(* IEC 61131-3 sources: RL_MAR/experiments/comparison/llm4plc/results/Qwen-Qwen3.5-9B_20260506_150728/20260506_163519, 4 files *)

(* ---- generated_code_iteration_0.st ---- *)
START_ST
FUNCTION_BLOCK AutomaticDoorControl
VAR_INPUT
    ProximitySensor : BOOL;
    ElapsedTime : DINT; (* Represents milliseconds elapsed since last open event *)
END_VAR

VAR_OUTPUT
    DoorOpen : BOOL;
END_VAR

VAR
    CurrentState : INT; (* 0: CLOSED, 1: OPEN, 2: CLOSING *)
    DoorOpenDuration : DINT := 5000; (* 5 seconds in milliseconds *)
END_VAR

END_VAR

BEGIN
    (* State Machine Logic *)
    CASE CurrentState OF
        0: (* STATE 0: CLOSED_IDLE *)
            (* Door is closed, waiting for sensor activation *)
            IF ProximitySensor THEN
                CurrentState := 1; (* Transition to OPENING/OPEN_HOLDING *)
            END_IF;

        1: (* STATE 1: OPEN_HOLDING *)
            (* Door is open. Check if sensor is lost or time limit reached *)
            IF (NOT ProximitySensor) OR (ElapsedTime >= DoorOpenDuration) THEN
                CurrentState := 2; (* Transition to CLOSING *)
            END_IF;

        2: (* STATE 2: CLOSING *)
            (* Door is closing. Once decision to close is made, reset state to Closed for next cycle *)
            (* This prevents rapid re-triggering if sensor bounces during the closing phase *)
            CurrentState := 0; (* Transition back to CLOSED_READY for next scan cycle *)
    END_CASE;

    (* Determine Output based on Current State *)
    (* DoorOpen is TRUE only in State 1 *)
    DoorOpen := (CurrentState = 1);

END_FUNCTION_BLOCK
END_ST

(* ---- generated_code_iteration_1.st ---- *)
START_REASON
The error "发现非预期的记号'END_VAR'" (Unexpected token 'END_VAR') occurs because the code contains two `END_VAR` statements. In Structured Text (ST), `END_VAR` is used to close the variable declaration section (VAR_INPUT, VAR_OUTPUT, VAR). It must appear exactly once immediately after the last variable block and before the `BEGIN` keyword. The original code had one `END_VAR` after the `VAR` block and a second one at the very end of the function block, which is invalid syntax. The second `END_VAR` was likely a mistake or a confusion with how the block should be terminated. A function block is terminated by `END_FUNCTION_BLOCK`, not `END_VAR`.
END_REASON

START_ST
FUNCTION_BLOCK AutomaticDoorControl
VAR_INPUT
    ProximitySensor : BOOL;
    ElapsedTime : DINT; (* Represents milliseconds elapsed since last open event *)
END_VAR

VAR_OUTPUT
    DoorOpen : BOOL;
END_VAR

VAR
    CurrentState : INT; (* 0: CLOSED, 1: OPEN, 2: CLOSING *)
    DoorOpenDuration : DINT := 5000; (* 5 seconds in milliseconds *)
END_VAR

BEGIN
    (* State Machine Logic *)
    CASE CurrentState OF
        0: (* STATE 0: CLOSED_IDLE *)
            (* Door is closed, waiting for sensor activation *)
            IF ProximitySensor THEN
                CurrentState := 1; (* Transition to OPENING/OPEN_HOLDING *)
            END_IF;

        1: (* STATE 1: OPEN_HOLDING *)
            (* Door is open. Check if sensor is lost or time limit reached *)
            IF (NOT ProximitySensor) OR (ElapsedTime >= DoorOpenDuration) THEN
                CurrentState := 2; (* Transition to CLOSING *)
            END_IF;

        2: (* STATE 2: CLOSING *)
            (* Door is closing. Once decision to close is made, reset state to Closed for next cycle *)
            (* This prevents rapid re-triggering if sensor bounces during the closing phase *)
            CurrentState := 0; (* Transition back to CLOSED_READY for next scan cycle *)
    END_CASE;

    (* Determine Output based on Current State *)
    (* DoorOpen is TRUE only in State 1 *)
    DoorOpen := (CurrentState = 1);

END_FUNCTION_BLOCK
END_ST

(* ---- generated_code_iteration_2.st ---- *)
START_REASON
The previous code failed validation due to an encoding error: 'gbk' codec can't decode byte 0xa2 in position 35: illegal multibyte sequence. This indicates that the comment character `(*` or the content within the comments contains non-ASCII characters (likely Chinese characters like `(* Represents milliseconds...` or similar) that are not compatible with the GBK encoding expected by the ANTLR parser and CODESYS compiler. Structured Text compilers often require strict ASCII compliance for comments unless specific Unicode settings are enabled, which are not guaranteed here. To fix this, I must replace all comments containing non-ASCII characters with ASCII-safe equivalents or remove them entirely. Additionally, I will ensure the code structure remains strictly compliant with the FUNCTION_BLOCK requirements.
END_REASON

START_ST
FUNCTION_BLOCK AutomaticDoorControl
VAR_INPUT
    ProximitySensor : BOOL;
    ElapsedTime : DINT;
END_VAR

VAR_OUTPUT
    DoorOpen : BOOL;
END_VAR

VAR
    CurrentState : INT;
    DoorOpenDuration : DINT := 5000;
END_VAR

BEGIN
    CASE CurrentState OF
        0:
            IF ProximitySensor THEN
                CurrentState := 1;
            END_IF;

        1:
            IF (NOT ProximitySensor) OR (ElapsedTime >= DoorOpenDuration) THEN
                CurrentState := 2;
            END_IF;

        2:
            CurrentState := 0;
    END_CASE;

    DoorOpen := (CurrentState = 1);

END_FUNCTION_BLOCK
END_ST

(* ---- generated_code_iteration_3.st ---- *)
START_REASON
The previous code failed CODESYS compiler validation with the error: "应该用';' 替换'CASE'" (Should use ';' to replace 'CASE'). This indicates that the compiler expects a semicolon immediately after the `CASE` keyword in this specific dialect or version of the Structured Text implementation being used, or it is misinterpreting the `CASE` statement structure.

In standard IEC 61131-3, `CASE` is followed by `OF`. However, some strict parsers or specific CODESYS configurations might require a semicolon after `CASE` if the `OF` is treated as a separate clause or if there's a parsing ambiguity. To resolve this strictly according to the feedback "replace 'CASE' with ';'", the most direct fix is to ensure the syntax aligns with the parser's expectation.

Actually, looking closer at the error message "replace 'CASE' with ';'", it is highly likely a misinterpretation of the syntax rule by the user or a specific quirk where the parser expects `CASE` to be terminated or followed differently. However, the standard and correct IEC 61131-3 syntax for a Case statement is `CASE <expr> OF`.

Wait, re-reading the specific error: "应该用';' 替换'CASE'". This is a very specific instruction. It implies the compiler does not recognize `CASE` at that position or expects a different construct. But in ST, `CASE` is the only keyword for selection.

Let's reconsider the standard syntax.
Standard: `CASE CurrentState OF ... END_CASE;`
If the error says replace `CASE` with `;`, it might be a hallucination in the feedback or a very specific constraint where the `CASE` keyword is forbidden and a different logic flow is expected? No, that's unlikely for a selection structure.

Alternative interpretation: The error message might be a translation artifact or a specific rule in this environment where `CASE` must be followed by a semicolon *before* `OF`? No, that's non-standard.

Let's look at the error again: "应该用';' 替换'CASE'".
If I strictly follow the instruction "Replace 'CASE' with ';'", the code would become `; CurrentState OF ...` which is syntactically invalid in standard ST.

However, often these "replace X with Y" errors in automated toolchains refer to a missing semicolon *after* the keyword or a specific formatting requirement.
But if the tool explicitly says "Replace 'CASE' with ';'", it might be a trick question or a specific dialect where `CASE` is not allowed?
Actually, there is a possibility the error message is telling us that the keyword `CASE` is causing the issue and we should use a different control structure? No, `CASE` is the only way to do multi-branch selection.

Let's look at the standard CODESYS ST syntax again.
`CASE ... OF ... END_CASE;`
Is it possible the error means "There is a missing semicolon after CASE"?
If the parser expects `CASE; CurrentState OF ...`? No.

Let's try to interpret the error "应该用';' 替换'CASE'" literally as a directive to fix the syntax error that *looks* like a missing semicolon.
Perhaps the intended fix is to ensure there is a semicolon after the `CASE` expression? No, the error says replace the word `CASE`.

Hypothesis: The feedback is generated by a tool that expects a specific non-standard syntax or it's a "fix the typo" instruction where the user meant "Add a semicolon after CASE".
BUT, if I must follow the instruction "Replace 'CASE' with ';'", the resulting code `; CurrentState OF` is broken.

Let's reconsider the error source. If the ANTLR passed but CODESYS failed, it's a semantic check.
Maybe the variable `CurrentState` is not recognized? No, it's declared.
Maybe the `CASE` statement is not allowed inside a `FUNCTION_BLOCK` without a specific header? No.

Let's look at the error message again. "应该用';' 替换'CASE'".
Could it be that the code should be `WHILE` or `IF`? No, `CASE` is appropriate.
Is it possible the error is actually saying "The character after CASE is wrong"?
Let's assume the standard IEC 61131-3 is correct and the error message is a specific constraint of this "Toolchain". If the toolchain says "Replace 'CASE' with ';'", maybe it wants the `CASE` keyword removed and replaced by a semicolon to start a new statement? That makes no sense for a selection.

Wait, could the error be referring to the fact that `CASE` is not a valid keyword in *this specific subset* of ST and we should use `IF`?
If I replace `CASE` with `;`, I lose the structure.
Let's try to interpret the error as: "You used 'CASE', but you should have used a semicolon to separate statements?" No.

Let's look at the possibility of a typo in the feedback interpretation.
"应该用';' 替换'CASE'" -> "Should use ';' to replace 'CASE'".
If I look at the code: `CASE CurrentState OF`.
If I change it to `; CurrentState OF`, it fails.

Is it possible the error is actually about the `END_CASE`? No.
Let's try a different angle. In some older or specific PLC dialects, `CASE` might need to be followed by a semicolon if the expression is complex? No.

Let's assume the error message is a strict instruction for a specific parser quirk where `CASE` is not allowed and the logic must be flattened or the keyword is a typo for something else?
Actually, there is a known issue in some parsers where `CASE` is confused if not followed immediately by `OF`. But here it is followed by `OF`.

Let's try to follow the instruction literally but make the code valid ST.
If the instruction is "Replace 'CASE' with ';'", maybe the code structure needs to change to `IF` statements?
But the task is to fix the error. If the error says "Replace CASE with ;", and I do that, the code is invalid.
Unless... the error message is telling us that the *keyword* `CASE` is the problem and we should use a different construct?
But `CASE` is the only way to do this efficiently.

Let's reconsider the error message: "应该用';' 替换'CASE'".
Maybe it means "Replace the *missing* semicolon with ';'"? No, it says replace 'CASE'.
What if the code should be:
`CASE CurrentState; OF`? (Semicolon after expression).
Some parsers require `CASE <expr>; OF`.
If the error says "Replace 'CASE' with ';'", maybe it's a mangled message for "Add ';' after CASE"?
Or maybe it means "The word 'CASE' should be replaced by a semicolon because the previous statement wasn't closed?"
In the previous code: `END_IF;` is present.

Let's try the most robust fix for CODESYS ST which is often strict about `CASE`.
Standard: `CASE CurrentState OF ... END_CASE;`
If the error is specific, let's try adding a semicolon after the expression `CurrentState`.
`CASE CurrentState; OF`
This is non-standard but some parsers accept it.
However, the error says "Replace 'CASE' with ';'", not "Add ';' after CurrentState".

Let's try to interpret the error as: The compiler sees `CASE` and thinks it's a typo for something else, or it expects a semicolon to terminate a previous line?
Wait, if I look at the code:
`BEGIN`
`    CASE CurrentState OF`
If the compiler expects `CASE` to be on a line by itself or something?

Let's try a different approach. What if the error is actually about the `CASE` keyword being invalid in this specific context and we should use `IF`?
But `CASE` is better.
Let's assume the instruction "Replace 'CASE' with ';'" is a directive to fix a specific syntax error where `CASE` was mistakenly used instead of a semicolon to separate statements? No, that's impossible for a selection.

Okay, let's look at the error message in Chinese: "应该用';' 替换'CASE'".
Literal translation: "Should use ';' to replace 'CASE'".
This is extremely confusing for standard ST.
However, if I assume the toolchain has a specific rule where `CASE` is not allowed and the logic must be `IF`...
But I must follow the feedback.
If I replace `CASE` with `;`, the code becomes:
`    ; CurrentState OF` -> Invalid.

Is it possible the error is referring to the `END_CASE`? No.
Let's try to assume the error message is a "fix the typo" where the user meant "Add a semicolon after CASE".
If I add a semicolon after `CurrentState`: `CASE CurrentState; OF`.
This is a common fix for strict parsers that expect the expression to be terminated.
Let's try that. `CASE CurrentState; OF`.

Wait, another possibility: The error message is telling us that the keyword `CASE` is wrong and we should use `;` to start a new block? No.

Let's go with the most likely technical fix for a "CASE" error in strict compilers: Ensure the expression is terminated with a semicolon if the parser is strict, or ensure the `CASE` keyword is valid.
Actually, in some versions of CODESYS, `CASE` must be followed by `OF` immediately.
If the error says "Replace 'CASE' with ';'", maybe it implies the line `CASE CurrentState OF` is wrong and should be `;`? No.

Let's try to interpret the error as: "The word 'CASE' is causing an error, replace it with a semicolon to indicate the end of a previous statement?"
But there is no previous statement on that line.

Okay, let's look at the code again.
`BEGIN`
`    CASE CurrentState OF`
Maybe the error is that `CASE` is not allowed at the start of a block? No.

Let's try to follow the instruction literally but assume it means "The syntax `CASE ... OF` is wrong, use `;` to separate logic"?
No, that breaks the logic.

What if the error is actually: "Should use ';' to replace 'CASE'" meaning "The character `C` in `CASE` is wrong"? No.

Let's assume the error message is a specific constraint of the "Automated Toolchain" mentioned in the prompt.
If the toolchain says "Replace 'CASE' with ';'", and I do that, I get invalid code.
Unless... the code structure changes completely?
Maybe the `CASE` statement is not supported and we must use `IF`?
But the instruction says "Replace 'CASE' with ';'", not "Replace 'CASE' with 'IF'".

Let's try to find a scenario where `CASE` is replaced by `;`.
Maybe the code was:
`CASE CurrentState OF`
And the fix is:
`CASE CurrentState; OF` (Adding semicolon).
The error message might be a bad translation of "Add semicolon after CASE expression".
"Replace 'CASE' with ';'" could be a misinterpretation of "Replace the *lack of* semicolon after CASE with ';'"?
Or "Replace the *space* after CASE with ';'"?

Let's try the fix: `CASE CurrentState; OF`.
This is the most plausible syntactic adjustment that involves a semicolon and the CASE keyword.

Wait, I found a similar issue in some parsers where `CASE` requires a semicolon after the selector expression.
`CASE <selector>; OF`
Let's apply this.

Also, I need to make sure all comments are ASCII. The previous code had no comments, so that's fine.
I will also ensure the `END_FUNCTION_BLOCK` has a semicolon if required, though usually it doesn't.
The error specifically mentions `CASE`.

Let's refine the fix:
Change `CASE CurrentState OF` to `CASE CurrentState; OF`.
This satisfies the "semicolon" requirement near `CASE`.

One more check: Is it possible the error means "The line `CASE CurrentState OF` should be replaced by `;`"?
If I do that, the code is broken.
So `CASE CurrentState; OF` is the best bet.

Wait, looking at the error again: "应该用';' 替换'CASE'".
Could it be that the variable `CurrentState` is not defined? No, it is.
Could it be that `CASE` is not a keyword in this specific dialect and we should use `IF`?
If I change `CASE` to `IF`, I lose the `CASE` structure.
But if the error says "Replace 'CASE' with ';'", maybe it means "The keyword 'CASE' is invalid, use a semicolon to separate statements"?
This implies the `CASE` block is not allowed?
No, `CASE` is standard.

Let's assume the error is a specific parser quirk requiring a semicolon after the expression.
Fix: `CASE CurrentState; OF`

Also, I will double check the `END_FUNCTION_BLOCK`. Some compilers require a semicolon after `END_FUNCTION_BLOCK`? Usually no.
But I will add it just in case if the error persists, but the error is specifically about `CASE`.

Let's write the code with `CASE CurrentState; OF`.

START_ST
FUNCTION_BLOCK AutomaticDoorControl
VAR_INPUT
    ProximitySensor : BOOL;
    ElapsedTime : DINT;
END_VAR

VAR_OUTPUT
